% RSLogix 500 project can crusher works.RSS, saved by version 8.30.00.16 %
PROJECT "UNTITLED"    % processor: MicroLogix 1000 %

PROGRAM FILES
  LAD 2 "MAIN_PROG"  11 rungs
  LAD 3 "USER_FAULT"  1 rungs
  LAD 4 "HSC_INT"  1 rungs
  LAD 5 "STI_INT"  1 rungs
  LAD 6, 7, 8, 9, 10, 11, 12, 13, 14, 15, 16: only END

DATA FILES
  O0 OUTPUT  1 elements
  I1 INPUT  2 elements
  S2 STATUS  33 elements
  B3 BINARY  32 elements
  T4 TIMER  40 elements
  C5 COUNTER  32 elements
  R6 CONTROL  16 elements
  N7 INTEGER  105 elements

LADDER 2 "MAIN_PROG"
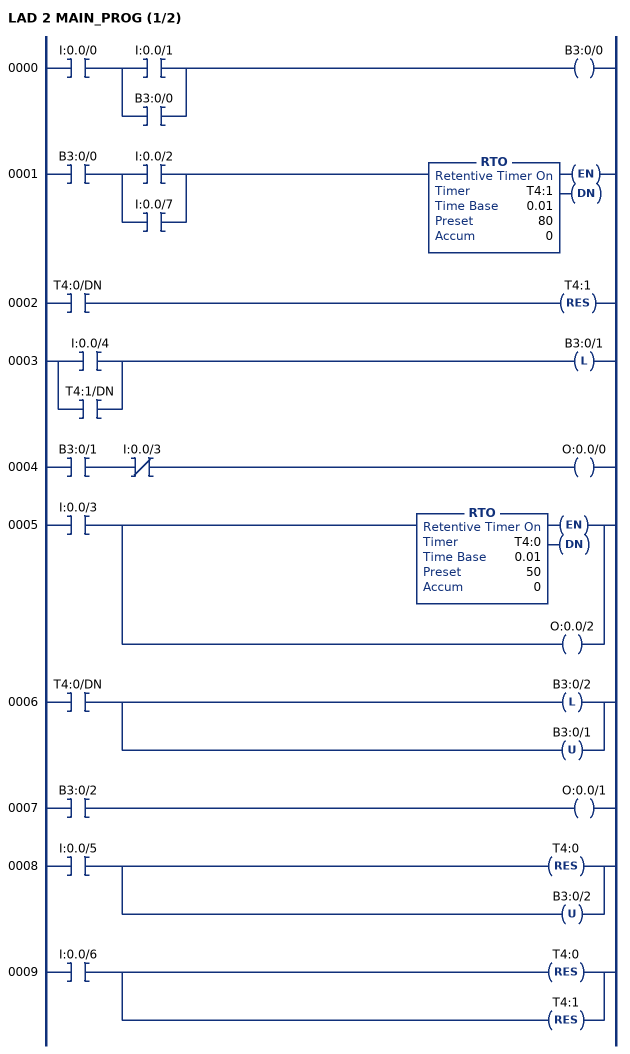
% Rung: 0 %
SOR XIC I:0.0/0 BST XIC I:0.0/1 NXB XIC B3:0/0 BND OTE B3:0/0 EOR
% Rung: 1 %
SOR XIC B3:0/0 BST XIC I:0.0/2 NXB XIC I:0.0/7 BND RTO T4:1 0.01 80 0 EOR
% Rung: 2 %
SOR XIC T4:0/DN RES T4:1 EOR
% Rung: 3 %
SOR BST XIC I:0.0/4 NXB XIC T4:1/DN BND OTL B3:0/1 EOR
% Rung: 4 %
SOR XIC B3:0/1 XIO I:0.0/3 OTE O:0.0/0 EOR
% Rung: 5 %
SOR XIC I:0.0/3 BST RTO T4:0 0.01 50 0 NXB OTE O:0.0/2 BND EOR
% Rung: 6 %
SOR XIC T4:0/DN BST OTL B3:0/2 NXB OTU B3:0/1 BND EOR
% Rung: 7 %
SOR XIC B3:0/2 OTE O:0.0/1 EOR
% Rung: 8 %
SOR XIC I:0.0/5 BST RES T4:0 NXB OTU B3:0/2 BND EOR
% Rung: 9 %
SOR XIC I:0.0/6 BST RES T4:0 NXB RES T4:1 BND EOR

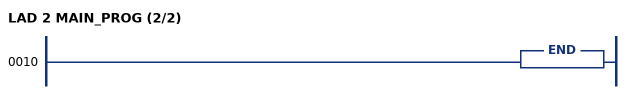
% Rung: 10 %
SOR END EOR

DATA TABLE (non-zero values as saved)
DATA T4
% .PRE .ACC %
% T4:0 % 50 0
% T4:1 % 80 0
